// global function to extract state identifier from combined value
FUNCTION f_GetState : uint
VAR_INPUT
  state     : UINT; // combined value of identifier + e_progress
END_VAR
VAR
END_VAR


IF (State > E_PROGRESS.PROGRESS_DONE)
THEN
  f_GetState        := state - E_PROGRESS.PROGRESS_DONE;

ELSIF (State > E_PROGRESS.PROGRESS_ERROR)
THEN
  f_GetState        := state - E_PROGRESS.PROGRESS_ERROR;

ELSIF (State > E_PROGRESS.PROGRESS_STILL_WORKING)
THEN
  f_GetState        := state - E_PROGRESS.PROGRESS_STILL_WORKING;

ELSIF (State > E_PROGRESS.PROGRESS_WORKING)
THEN
  f_GetState        := state - E_PROGRESS.PROGRESS_WORKING;

ELSIF (State > E_PROGRESS.PROGRESS_OCCUPIED)
THEN
  f_GetState        := state - E_PROGRESS.PROGRESS_OCCUPIED;

ELSIF (State > E_PROGRESS.PROGRESS_CHECK)
THEN
  f_GetState        := state - E_PROGRESS.PROGRESS_CHECK;

ELSIF (State > E_PROGRESS.PROGRESS_STARTUP)
THEN
  f_GetState        := state - E_PROGRESS.PROGRESS_STARTUP;

ELSIF (State > E_PROGRESS.PROGRESS_PREPARE)
THEN
  f_GetState        := state - E_PROGRESS.PROGRESS_DONE;

ELSIF (State > E_PROGRESS.PROGRESS_BUSY)
THEN
  f_GetState        := state - E_PROGRESS.PROGRESS_BUSY;

ELSIF (State > E_PROGRESS.PROGRESS_INIT)
THEN
  f_GetState        := state - E_PROGRESS.PROGRESS_INIT;

ELSE
  f_GetState        := state;
END_IF

END_FUNCTION

(* stored: Version 1.1.0.1, ProductVersion 3.1.4024.12
   POU f_GetState: Id {865f2491-fb88-41b7-a624-10aefc803067}, SpecialFunc None *)
